INTERFACE I_MotionTask EXTENDS I_Cyclic, I_TaskResult, I_Command

PROPERTY Axis : I_Axis
GET
END_GET
SET
END_SET
END_PROPERTY

{attribute 'monitoring' := 'call'}
PROPERTY Name : T_MaxString
GET
END_GET
SET
END_SET
END_PROPERTY

END_INTERFACE

(* stored: Version 1.1.0.1, ProductVersion 3.1.4026.18
   Itf I_MotionTask: Id {d5273dc3-25ad-4a63-8b13-a40daf64efb7}
   Property Axis: Id {4753dee2-dbdc-4624-b8ac-55f4639e77da}
   Get Get: Id {84c026c1-eb86-4df7-9177-a1a207ef85b1}
   Set Set: Id {81ac9302-32be-4d4f-a811-6b294bbb4929}
   Property Name: Id {ec35e34f-483a-4d12-82eb-73d25abaa418}
   Get Get: Id {72723fa9-23c4-450f-9b14-9f574d0ed054}
   Set Set: Id {1e43d782-3416-4b4c-adfc-427782c52171} *)
